FUNCTION_BLOCK SplitInitEv (* Template for a simple Basic Function Block Type *)
  (* Standard: 61499-2 *)
  (* Version 1.0, 2020-03-21, Duc Do Tran, OFFIS e.V. *)
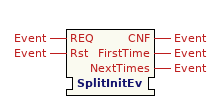
  EVENT_INPUT
    REQ; (* Normal Execution Request *)
    Rst;
  END_EVENT
  EVENT_OUTPUT
    CNF; (* Execution Confirmation *)
    FirstTime; (* Initialization Confirm *)
    NextTimes;
  END_EVENT
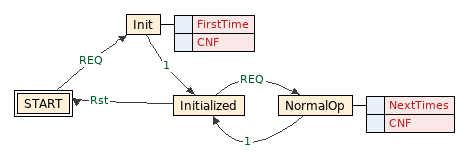
  EC_STATES
    START; (* Initial State *)
    Init : -> FirstTime, -> CNF; (* Initialization *)
    NormalOp : -> NextTimes, -> CNF; (* Normal execution *)
    Initialized;
  END_STATES
  EC_TRANSITIONS
    Init TO Initialized := 1;
    Initialized TO NormalOp := REQ;
    Initialized TO START := Rst;
    NormalOp TO Initialized := 1;
    START TO Init := REQ;
  END_TRANSITIONS
END_FUNCTION_BLOCK
